SUBAPPLICATION GreenWhiteBackground3_AX (* Hintergrundfarbe (TRUE -> Grün, FALSE -> Weiß) für 3 Objekte (AX-Adapter) *)
  (* Standard: 61499-2 *)
  (* Version 1.0, 2022-11-10, Franz Höpfinger, Meisterschulen am Ostbahnhof *)
  PACKAGE MyLib::sys;
  IMPORT isobus::UT::Q::const::IDs::ID_NULL;
  IMPORT isobus::UT::Q::const::colours::COLOR_WHITE;
  IMPORT isobus::UT::Q::const::colours::COLOR_GREEN;
  (* Documentation:
  Hintergrundfarbe für ein normales VT-Objekt UND ein Auxiliary-Function-Objekt gemeinsam
   Setzt aus einem einzigen DI1-Eingang (und einem gemeinsamen Farb-Select) die Hintergrundfarbe (TRUE -> Grün, FALSE -> Weiß) für zwei unterschiedliche Objekte gleichzeitig:
    - u16ObjId: ein normales VT-Objekt (z.B. SoftKey) - ein Q_BackgroundColour-Kommando ans VT.
   - u16ObjIdA: ein Auxiliary-Function-Type-2-Objekt (Object-ID-Bereich 31000–31999) - wie bei GreenWhiteBackground2_AX zwei Kommandos (Q_BackgroundColour ans VT für die Vorschau, Q_BackgroundColourAux ans Aux-Handle selbst).
    Insgesamt also drei Kommandos (daher der Name) aus einer einzigen, gemeinsamen Farbauswahl - gedacht für den Fall, dass ein normales VT-Objekt (z.B. SoftKey) und ein Aux-Objekt (z.B. Joystick) dieselbe Funktion auslösen und ihr Feedback synchron zeigen sollen (siehe Uebung_010f3_AX). Für nur ein normales Objekt GreenWhiteBackground1_AX, für nur ein Aux-Objekt GreenWhiteBackground2_AX verwenden - nicht beide einzeln kombinieren, wenn GreenWhiteBackground3_AX den Fall bereits abdeckt (siehe Uebung_010f4_AX als Negativbeispiel dafür).
  *)
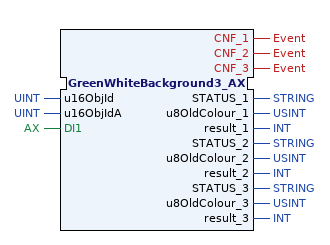
  EVENT_OUTPUT
    CNF_1;
    CNF_2;
    CNF_3;
  END_EVENT
  VAR_INPUT
    u16ObjId : UINT := ID_NULL; (* Object ID Softkey *)
    u16ObjIdA : UINT := ID_NULL; (* Object ID AUX *)
  END_VAR
  VAR_OUTPUT
    STATUS_1 : STRING; (* Service Status *)
    u8OldColour_1 : USINT; (* Old value of ID *)
    result_1 : INT; (* retval see description *)
    STATUS_2 : STRING; (* Service Status *)
    u8OldColour_2 : USINT; (* Old value of ID *)
    result_2 : INT; (* retval see description *)
    STATUS_3 : STRING; (* Service Status *)
    u8OldColour_3 : USINT; (* Old value of ID *)
    result_3 : INT; (* retval see description *)
  END_VAR
  SOCKETS
    DI1 : adapter::types::unidirectional::AX; (* Selector *)
  END_SOCKETS
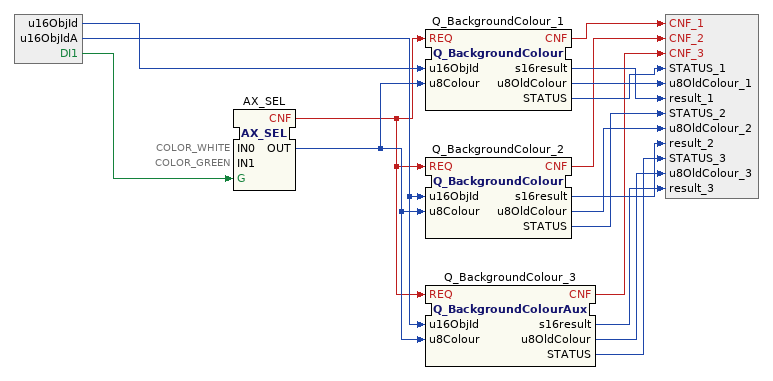
  FBS
    Q_BackgroundColour_1 : isobus::UT::Q::Q_BackgroundColour;
    Q_BackgroundColour_2 : isobus::UT::Q::Q_BackgroundColour;
    Q_BackgroundColour_3 : isobus::UT::Q::Q_BackgroundColourAux;
    AX_SEL : adapter::iec61131::selection::AX_SEL(IN0 := COLOR_WHITE, IN1 := COLOR_GREEN);
  END_FBS
  EVENT_CONNECTIONS
    Q_BackgroundColour_1.CNF TO CNF_1;
    Q_BackgroundColour_2.CNF TO CNF_2;
    Q_BackgroundColour_3.CNF TO CNF_3;
    AX_SEL.CNF TO Q_BackgroundColour_1.REQ;
    AX_SEL.CNF TO Q_BackgroundColour_2.REQ;
    AX_SEL.CNF TO Q_BackgroundColour_3.REQ;
  END_CONNECTIONS
  DATA_CONNECTIONS
    u16ObjId TO Q_BackgroundColour_1.u16ObjId;
    Q_BackgroundColour_1.s16result TO result_1;
    Q_BackgroundColour_1.u8OldColour TO u8OldColour_1;
    Q_BackgroundColour_1.STATUS TO STATUS_1;
    AX_SEL.OUT TO Q_BackgroundColour_1.u8Colour;
    u16ObjIdA TO Q_BackgroundColour_2.u16ObjId;
    Q_BackgroundColour_2.s16result TO result_2;
    Q_BackgroundColour_2.u8OldColour TO u8OldColour_2;
    Q_BackgroundColour_2.STATUS TO STATUS_2;
    AX_SEL.OUT TO Q_BackgroundColour_2.u8Colour;
    u16ObjIdA TO Q_BackgroundColour_3.u16ObjId;
    Q_BackgroundColour_3.s16result TO result_3;
    Q_BackgroundColour_3.u8OldColour TO u8OldColour_3;
    Q_BackgroundColour_3.STATUS TO STATUS_3;
    AX_SEL.OUT TO Q_BackgroundColour_3.u8Colour;
  END_CONNECTIONS
  ADAPTER_CONNECTIONS
    DI1 TO AX_SEL.G;
  END_CONNECTIONS
END_SUBAPPLICATION
